(* CODESYS project SLL_IFM_CRXXXX_exported_from_plc.library
   Author: adam@sperrinlogic.com
   Version: 0.0.0.1
   Title: SLL_IFM_CRXXXX
   DefaultNamespace: SLL_IFM_CRXXXX
   Placeholder: SLL_IFM_CRXXXX
   Company: SLL

Project tree, tasks and I/O mapping:
  libraries: Util, 3.5.19.0 (System); Standard, 3.5.18.0 (System); ifmTypes, 1.9.6.0 (ifm electronic); ifmRawCAN, 4.0.3.0 (ifm electronic); ifmDeviceCR07nn, 1.2.2.0 (ifm electronic); SysTime, 3.5.17.0 (System); ifmIOcommon, 2.4.0.0 (ifm electronic); CmpSchedule, 3.5.17.0 (System); SysTypes Interfaces, * (System); SysTypes2 Interfaces, * (System); CmpIecTask, 3.5.19.0 (System); CmpErrors2 Interfaces, * (System); CmpErrors, 3.3.1.40 (System); SysFileAsync, 3.5.19.0 (System); SysTypes, 3.1.2.0 (System); SLL Common, 0.0.0.1 (SLL)
  Library Information/
    function IsLibReleased [ST]
    function GetLibVersionNumber [ST]
    function GetLibVersion [ST]
  data type PLC_CRXXXX_CAN_Status
  program PLC_CRXXXX_System_Udp [FBD]
  data type IFM_CRXXXX_System_STRUCT
  function block UDP_RX_CHECK_HB_FB [FBD]
  data type UDP_RX_STATS_HB_STRUCT
  data type IFM_HMI_Version_System_Header
  function block Get_Task_Info [ST]
  data type PLC_TASK_INFO_STRUCT
  program PLC_CRXXXX_System [FBD]
*)

// PLC_CRXXXX_CAN_Status
TYPE PLC_CRXXXX_CAN_Status :
STRUCT
	xError: BOOL;
	eDiagInfo: ifmTypes.DIAG_INFO;
	eBaudrate: ifmDevice.CAN_BAUDRATE;
	eBusState: ifmRCAN.BUS_STATE;
	uiErrorCntRx: UINT;
	uiErrorCntTx: UINT;
	xWarningRx: BOOL;
	xWarningTx: BOOL;
	udiCountRx: UDINT;
	usiBusLoad: USINT;
END_STRUCT
END_TYPE

// IFM_CRXXXX_System_STRUCT
TYPE IFM_CRXXXX_System_STRUCT :
STRUCT
	CycleCounter:DWORD;
	CycleFreq:REAL;
	CycleSecCounter:DWORD;
	CycleSecFreq:REAL;
	UpTimeMs:DWORD;
	VBB15_mV:UINT;
	VBB30_mV:UINT;
	PCB_Temp:INT;
	CPU_Temp:INT;
	TaskInfo: PLC_TASK_INFO_STRUCT;
	CAN0: PLC_CRXXXX_CAN_Status;
	CAN1: PLC_CRXXXX_CAN_Status;
	CAN2: PLC_CRXXXX_CAN_Status;
	CAN3: PLC_CRXXXX_CAN_Status;	
END_STRUCT
END_TYPE

// UDP_RX_STATS_HB_STRUCT
TYPE UDP_RX_STATS_HB_STRUCT :
STRUCT
	PLC_UpTimeMs:DINT;
	PLC_UpTimeMs_Last: DINT;
	PLC_UpTimeMs_Diff: DINT;
	
	Max_Diff_Value: DINT;	

	Error_LT_Count: DINT;
	Error_Diff_Count: DINT;
	Error_Frozen_Count: DINT;

	Warn_LT_Count: DINT;
	
	Warn_Diff_Count: DINT;
	Warn_Diff_TimeStamp: DWORD;
	Warn_Diff_Since: DWORD;

	Warn_Frozen_Count: DINT;

	Warn_Frozen_TimeStamp: DWORD;
	Warn_Frozen_Since: DWORD;	
END_STRUCT
END_TYPE

// IFM_HMI_Version_System_Header
TYPE IFM_HMI_Version_System_Header :
STRUCT
	TickMs: DWORD;
	Version_String: STRING(20);
	Version_Nums: ARRAY [0..3] OF WORD; 
	IO_Flags: WORD; // future use? special modes?
END_STRUCT
END_TYPE

// PLC_TASK_INFO_STRUCT
TYPE PLC_TASK_INFO_STRUCT :
STRUCT
    dwCycleTimeMainTask: DWORD;       
    dwCycleTimeSecTask: DWORD;       
    dwIntervalMainTask: DWORD;
    dwIntervalSecTask: DWORD;
    fMainTaskCpuLoad: REAL;
    fSecTaskCpuLoad: REAL;
    sNameMainTask: STRING(20);	
    sNameSecTask: STRING(20);	
END_STRUCT
END_TYPE

// Library Information/IsLibReleased
// This function has been automatically generated from the project information.
FUNCTION IsLibReleased : BOOL
VAR_INPUT
	
END_VAR

IsLibReleased := FALSE;

END_FUNCTION

// Library Information/GetLibVersionNumber
// This function has been automatically generated from the project information.
FUNCTION GetLibVersionNumber : DWORD
VAR_INPUT
	
END_VAR

GetLibVersionNumber := 1;

END_FUNCTION

// Library Information/GetLibVersion
// This function has been automatically generated from the project information.
FUNCTION GetLibVersion : VERSION
VAR_INPUT
	
END_VAR

GetLibVersion.uiMajor := 0;
GetLibVersion.uiMinor := 0;
GetLibVersion.uiServicePack := 0;
GetLibVersion.uiPatch := 1;

END_FUNCTION

// PLC_CRXXXX_System_Udp
PROGRAM PLC_CRXXXX_System_Udp

VAR_INPUT
	System: REFERENCE TO IFM_CRXXXX_System_STRUCT;
END_VAR

VAR	
	Cycle_Freq_FB: Cycle_Freq_REAL;
END_VAR

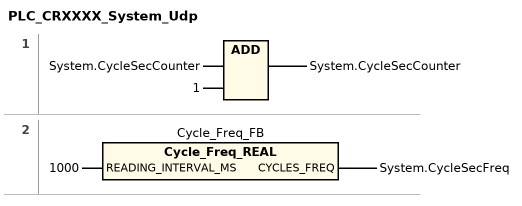
// NETWORK 1
System.CycleSecCounter := System.CycleSecCounter + 1;

// NETWORK 2
Cycle_Freq_FB(READING_INTERVAL_MS := 1000); // Cycle_Freq_REAL
System.CycleSecFreq := Cycle_Freq_FB.CYCLES_FREQ;

END_PROGRAM

// UDP_RX_CHECK_HB_FB
FUNCTION_BLOCK UDP_RX_CHECK_HB_FB
VAR_INPUT
	RESET: BOOL;	
	RESET_STATS: BOOL;
	RESET_ALARMS:BOOL;
	PlcTimeMs_Ip: DWORD;
	Moniotoring_Start_ms: DINT;	
	Warning_Diff_ms:DINT;
	Warning_Frozen_ms:DINT;
	Error_Diff_ms: DINT;
	Error_Frozen_ms: DINT;
	Error_Missing_ms: DINT;
	Error_Recovery_ms:DINT;
END_VAR
VAR_OUTPUT
	Monitoring: BOOL;	
	CommsError: BOOL;	
	Error_Missing: BOOL;
	Error_LessThan: BOOL;
	Error_Diff: BOOL;
	Error_Frozen: BOOL;
	Warning_Diff:BOOL;
	Warning_Frozen:BOOL;
	Unavail:BOOL:=TRUE;
END_VAR
VAR	
	TickMs: DWORD;
	TickMsWarmInit: DWORD;	
	
	RESET_Timestamp: DWORD;	
	RESET_Since_Ms: DWORD;
	
	Warning_Duration_Ms:DWORD:=1000;
	
	Warn_Frozen_TON:TON;
	
	Error_Missing_Active:BOOL;
	Error_Missing_Active_TON: TON;
	Error_Missing_SR: SR;
	Error_Missing_Reset_TON: TON;	
	Error_Missing_Set_TON: TON;
	
	Error_Frozen_Active: BOOL;
	Error_Frozen_Active_TON: TON;	
	Error_Frozen_SR: SR;
	Error_Frozen_Reset_TON: TON;
	Error_Frozen_Set_TON: TON;
	
	Error_Diff_Active: BOOL;
	Error_Diff_SR: SR;
	Error_Diff_Reset_TON: TON;
	Error_Diff_Set_TON: TON;
	
	Error_LessThan_Active: BOOL;
	Error_LessThan_SR: SR;
	Error_LessThan_Reset_TON: TON;	
	Error_LessThan_Set_TON: TON;
	Reset_Idle_TOF: TOF;
END_VAR

VAR_IN_OUT
	STATS: UDP_RX_STATS_HB_STRUCT;	
END_VAR
VAR // added by the converter: edge detectors and wires of the graphical bodies
    _w1, _w2 : BOOL;
    _rt1, _rt2, _rt3 : R_TRIG;
END_VAR

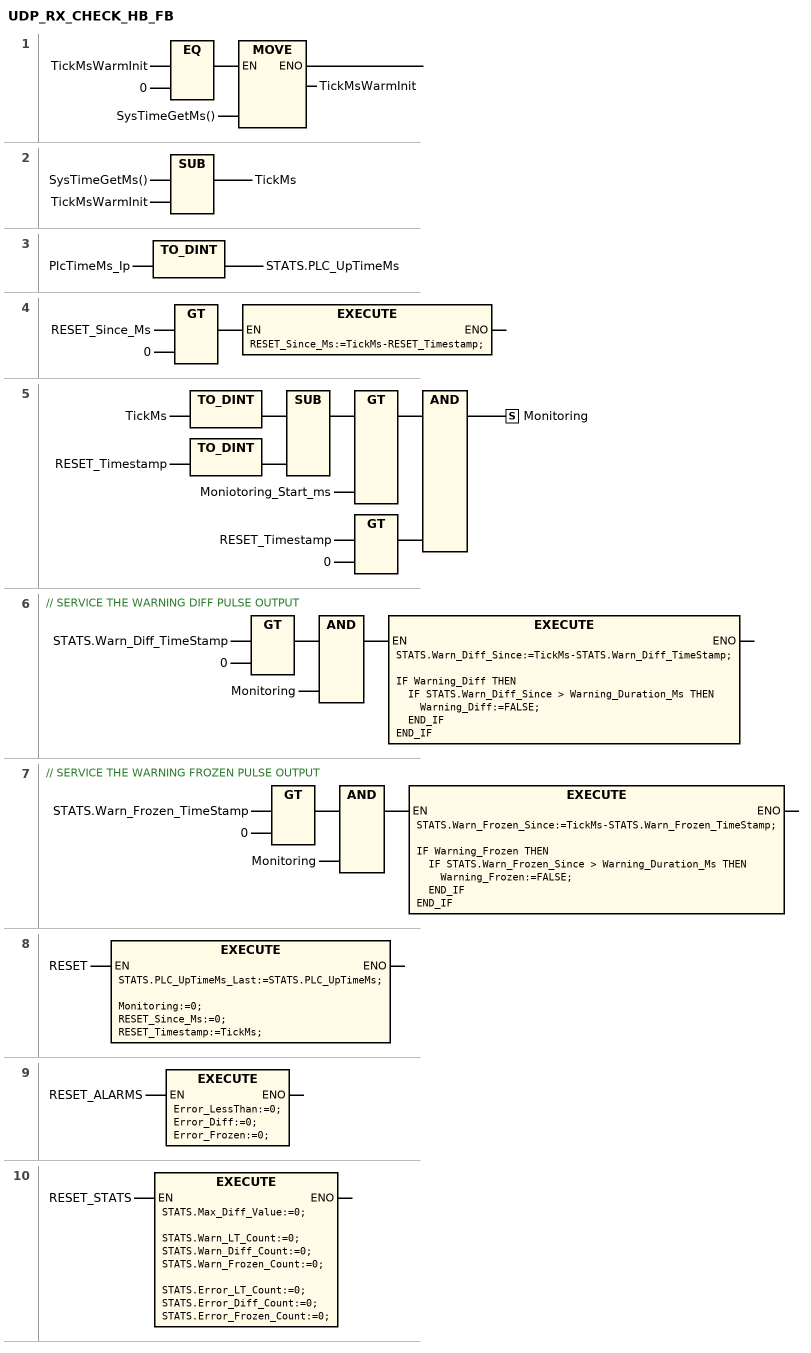
// NETWORK 1
IF TickMsWarmInit = 0 THEN TickMsWarmInit := SysTimeGetMs(); END_IF

// NETWORK 2
TickMs := (SysTimeGetMs()) - TickMsWarmInit;

// NETWORK 3
STATS.PLC_UpTimeMs := TO_DINT(PlcTimeMs_Ip);

// NETWORK 4
IF RESET_Since_Ms > 0 THEN RESET_Since_Ms:=TickMs-RESET_Timestamp; END_IF

// NETWORK 5
Monitoring S= TO_DINT(TickMs) - TO_DINT(RESET_Timestamp) > Moniotoring_Start_ms AND RESET_Timestamp > 0;

// NETWORK 6
// // SERVICE THE WARNING DIFF PULSE OUTPUT
IF STATS.Warn_Diff_TimeStamp > 0 AND Monitoring THEN
    STATS.Warn_Diff_Since:=TickMs-STATS.Warn_Diff_TimeStamp;
    
    IF Warning_Diff THEN
    	IF STATS.Warn_Diff_Since > Warning_Duration_Ms THEN
    		Warning_Diff:=FALSE;
    	END_IF
    END_IF
END_IF

// NETWORK 7
// // SERVICE THE WARNING FROZEN PULSE OUTPUT
IF STATS.Warn_Frozen_TimeStamp > 0 AND Monitoring THEN
    STATS.Warn_Frozen_Since:=TickMs-STATS.Warn_Frozen_TimeStamp;
    
    IF Warning_Frozen THEN
    	IF STATS.Warn_Frozen_Since > Warning_Duration_Ms THEN
    		Warning_Frozen:=FALSE;
    	END_IF
    END_IF
END_IF

// NETWORK 8
IF RESET THEN
    STATS.PLC_UpTimeMs_Last:=STATS.PLC_UpTimeMs;
    
    Monitoring:=0;
    RESET_Since_Ms:=0;
    RESET_Timestamp:=TickMs;
END_IF

// NETWORK 9
IF RESET_ALARMS THEN
    Error_LessThan:=0;
    Error_Diff:=0;
    Error_Frozen:=0;
END_IF

// NETWORK 10
IF RESET_STATS THEN
    STATS.Max_Diff_Value:=0;
    
    STATS.Warn_LT_Count:=0;
    STATS.Warn_Diff_Count:=0;
    STATS.Warn_Frozen_Count:=0;
    
    STATS.Error_LT_Count:=0;
    STATS.Error_Diff_Count:=0;
    STATS.Error_Frozen_Count:=0;
END_IF

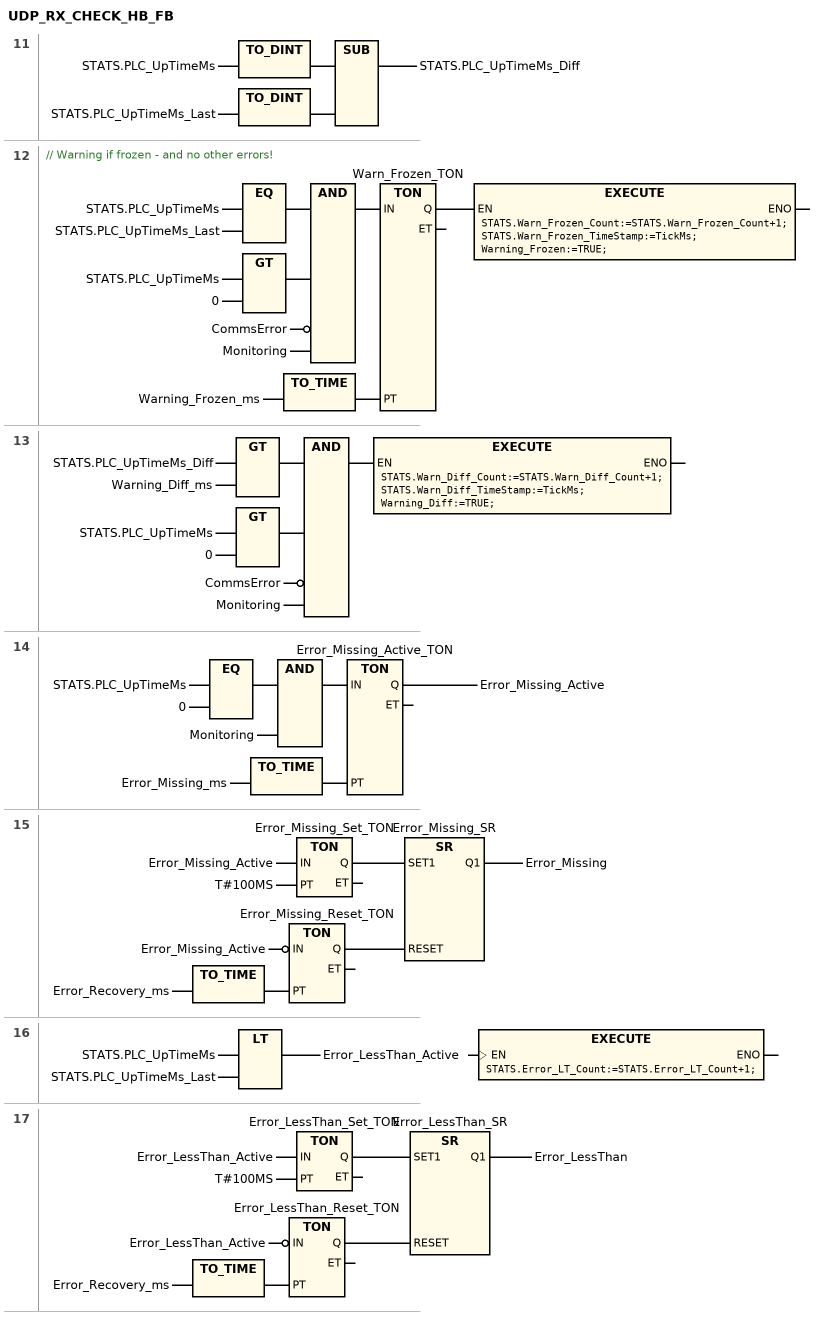
// NETWORK 11
STATS.PLC_UpTimeMs_Diff := TO_DINT(STATS.PLC_UpTimeMs) - TO_DINT(STATS.PLC_UpTimeMs_Last);

// NETWORK 12
// // Warning if frozen - and no other errors!
Warn_Frozen_TON(IN := STATS.PLC_UpTimeMs = STATS.PLC_UpTimeMs_Last AND STATS.PLC_UpTimeMs > 0 AND NOT CommsError AND Monitoring, PT := TO_TIME(Warning_Frozen_ms)); // TON
IF Warn_Frozen_TON.Q THEN
    STATS.Warn_Frozen_Count:=STATS.Warn_Frozen_Count+1;
    STATS.Warn_Frozen_TimeStamp:=TickMs;
    Warning_Frozen:=TRUE;
END_IF

// NETWORK 13
IF STATS.PLC_UpTimeMs_Diff > Warning_Diff_ms AND STATS.PLC_UpTimeMs > 0 AND NOT CommsError AND Monitoring THEN
    STATS.Warn_Diff_Count:=STATS.Warn_Diff_Count+1;
    STATS.Warn_Diff_TimeStamp:=TickMs;
    Warning_Diff:=TRUE;
END_IF

// NETWORK 14
Error_Missing_Active_TON(IN := STATS.PLC_UpTimeMs = 0 AND Monitoring, PT := TO_TIME(Error_Missing_ms)); // TON
Error_Missing_Active := Error_Missing_Active_TON.Q;

// NETWORK 15
Error_Missing_Set_TON(IN := Error_Missing_Active, PT := T#100MS); // TON
Error_Missing_Reset_TON(IN := NOT Error_Missing_Active, PT := TO_TIME(Error_Recovery_ms)); // TON
Error_Missing_SR(SET1 := Error_Missing_Set_TON.Q, RESET := Error_Missing_Reset_TON.Q); // SR
Error_Missing := Error_Missing_SR.Q1;

// NETWORK 16
_w1 := STATS.PLC_UpTimeMs < STATS.PLC_UpTimeMs_Last;
Error_LessThan_Active := _w1;
_rt1(CLK := _w1);
IF _rt1.Q THEN STATS.Error_LT_Count:=STATS.Error_LT_Count+1; END_IF

// NETWORK 17
Error_LessThan_Set_TON(IN := Error_LessThan_Active, PT := T#100MS); // TON
Error_LessThan_Reset_TON(IN := NOT Error_LessThan_Active, PT := TO_TIME(Error_Recovery_ms)); // TON
Error_LessThan_SR(SET1 := Error_LessThan_Set_TON.Q, RESET := Error_LessThan_Reset_TON.Q); // SR
Error_LessThan := Error_LessThan_SR.Q1;

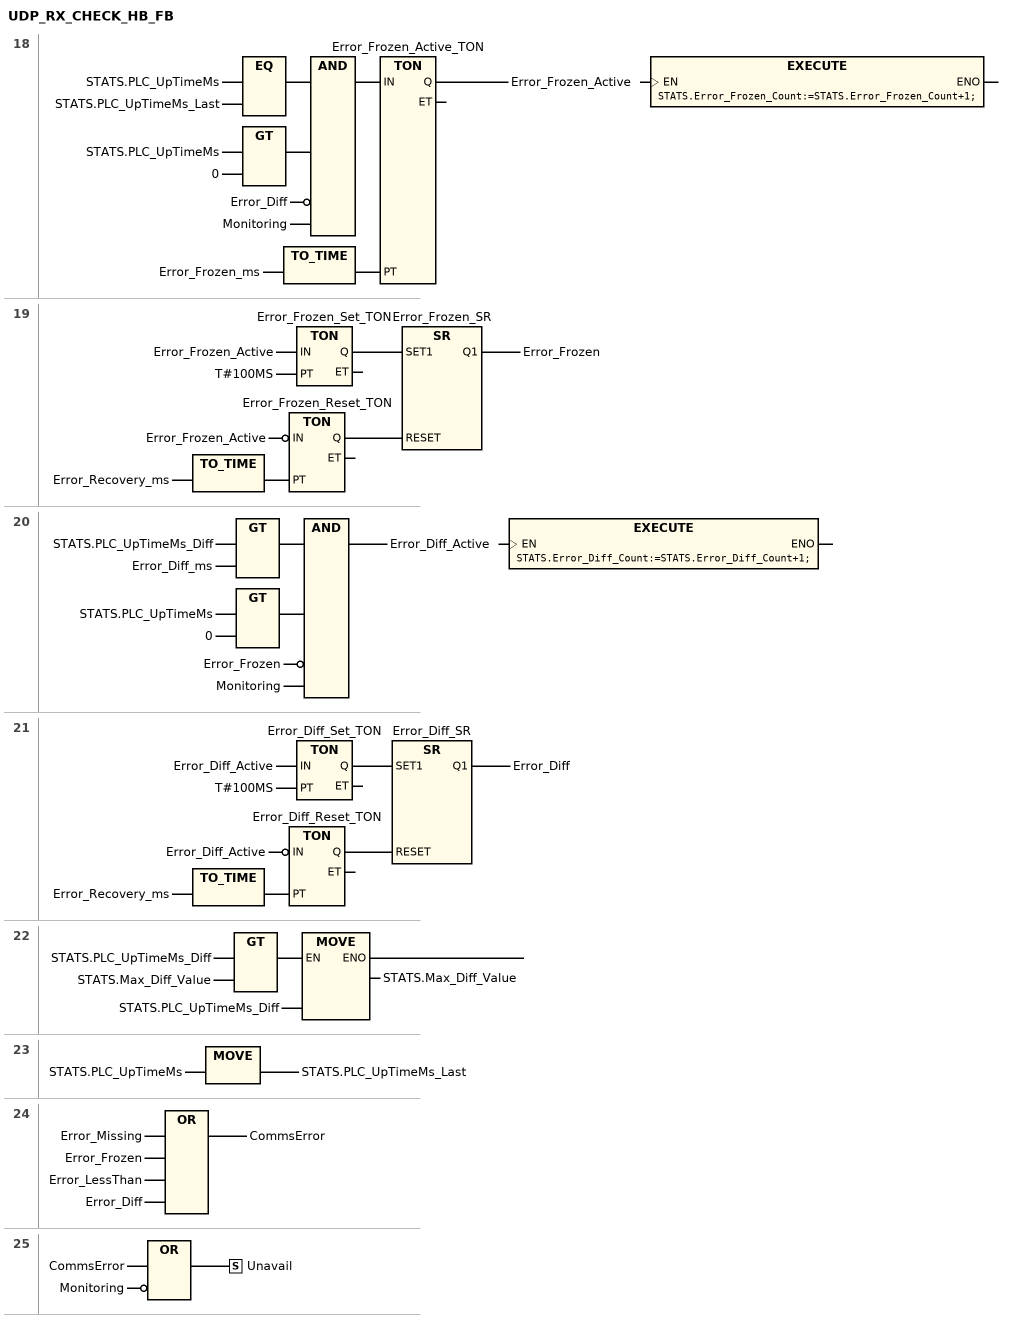
// NETWORK 18
Error_Frozen_Active_TON(IN := STATS.PLC_UpTimeMs = STATS.PLC_UpTimeMs_Last AND STATS.PLC_UpTimeMs > 0 AND NOT Error_Diff AND Monitoring, PT := TO_TIME(Error_Frozen_ms)); // TON
Error_Frozen_Active := Error_Frozen_Active_TON.Q;
_rt2(CLK := Error_Frozen_Active_TON.Q);
IF _rt2.Q THEN STATS.Error_Frozen_Count:=STATS.Error_Frozen_Count+1; END_IF

// NETWORK 19
Error_Frozen_Set_TON(IN := Error_Frozen_Active, PT := T#100MS); // TON
Error_Frozen_Reset_TON(IN := NOT Error_Frozen_Active, PT := TO_TIME(Error_Recovery_ms)); // TON
Error_Frozen_SR(SET1 := Error_Frozen_Set_TON.Q, RESET := Error_Frozen_Reset_TON.Q); // SR
Error_Frozen := Error_Frozen_SR.Q1;

// NETWORK 20
_w2 := STATS.PLC_UpTimeMs_Diff > Error_Diff_ms AND STATS.PLC_UpTimeMs > 0 AND NOT Error_Frozen AND Monitoring;
Error_Diff_Active := _w2;
_rt3(CLK := _w2);
IF _rt3.Q THEN STATS.Error_Diff_Count:=STATS.Error_Diff_Count+1; END_IF

// NETWORK 21
Error_Diff_Set_TON(IN := Error_Diff_Active, PT := T#100MS); // TON
Error_Diff_Reset_TON(IN := NOT Error_Diff_Active, PT := TO_TIME(Error_Recovery_ms)); // TON
Error_Diff_SR(SET1 := Error_Diff_Set_TON.Q, RESET := Error_Diff_Reset_TON.Q); // SR
Error_Diff := Error_Diff_SR.Q1;

// NETWORK 22
IF STATS.PLC_UpTimeMs_Diff > STATS.Max_Diff_Value THEN STATS.Max_Diff_Value := STATS.PLC_UpTimeMs_Diff; END_IF

// NETWORK 23
STATS.PLC_UpTimeMs_Last := STATS.PLC_UpTimeMs;

// NETWORK 24
CommsError := Error_Missing OR Error_Frozen OR Error_LessThan OR Error_Diff;

// NETWORK 25
Unavail S= CommsError OR NOT Monitoring;

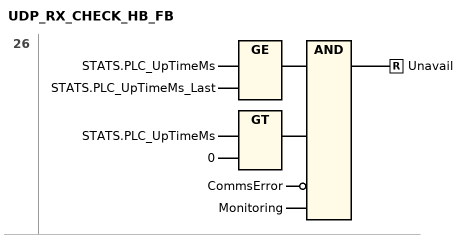
// NETWORK 26
Unavail R= STATS.PLC_UpTimeMs >= STATS.PLC_UpTimeMs_Last AND STATS.PLC_UpTimeMs > 0 AND NOT CommsError AND Monitoring;

END_FUNCTION_BLOCK

// Get_Task_Info
FUNCTION_BLOCK Get_Task_Info
VAR_INPUT
	sample_rate_tm:DWORD:=500;
END_VAR
VAR
    hFirstTask, hSecTask                       :    SysTypes.RTS_IEC_HANDLE;
    iecResult                                  :    SysTypes.RTS_IEC_RESULT;
    sAppName                                   :    STRING := 'Application';
    pIecInfo                                   :    POINTER TO CmpIecTask.Task_Info2;
	
	last_sample_ms: DWORD;
	diff_ms: DWORD;	
END_VAR

VAR_OUTPUT
	TaskInfo: PLC_TASK_INFO_STRUCT;
END_VAR

diff_ms := SysTimeGetMs() - last_sample_ms;

IF diff_ms < sample_rate_tm THEN
	RETURN;
END_IF

hFirstTask := CmpIecTask.IecTaskGetFirst(pszAppName := ADR(sAppName), pResult := ADR(iecResult));

IF ((hFirstTask <> SysTypes.RTS_INVALID_HANDLE) AND (iecResult = CmpErrors.Errors.ERR_OK)) THEN
    pIecInfo := CmpIecTask.IecTaskGetInfo3(hIecTask := hFirstTask, pResult := ADR(iecResult));
    TaskInfo.dwIntervalMainTask := pIecInfo^.dwInterval;
    TaskInfo.dwCycleTimeMainTask := pIecInfo^.dwCycleTime;
    TaskInfo.sNameMainTask := pIecInfo^.pszName^;
	
    hSecTask := IecTaskGetNext(pszAppName := ADR(sAppName), hPrevIecTask := hFirstTask, pResult := ADR(iecResult));
    IF ((hSecTask <> SysTypes.RTS_INVALID_HANDLE) AND (iecResult = CmpErrors.Errors.ERR_OK)) THEN
        pIecInfo := CmpIecTask.IecTaskGetInfo3(hIecTask := hSecTask, pResult := ADR(iecResult));
        TaskInfo.dwIntervalSecTask := pIecInfo^.dwInterval;
        TaskInfo.dwCycleTimeSecTask := pIecInfo^.dwCycleTime;
        TaskInfo.sNameSecTask := pIecInfo^.pszName^;
    END_IF
END_IF

TaskInfo.fMainTaskCpuLoad:=TO_REAL(TaskInfo.dwCycleTimeMainTask*100)/TO_REAL(TaskInfo.dwIntervalMainTask);
TaskInfo.fSecTaskCpuLoad:=TO_REAL(TaskInfo.dwCycleTimeSecTask*100)/TO_REAL(TaskInfo.dwIntervalSecTask);

END_FUNCTION_BLOCK

// PLC_CRXXXX_System
PROGRAM PLC_CRXXXX_System

VAR_INPUT
	System: REFERENCE TO IFM_CRXXXX_System_STRUCT;
END_VAR

VAR	
	Temperature_PCB_FB: ifmIOcommon.Temperature;
	Temperature_CPU_FB: ifmIOcommon.Temperature;	
	SystemSupply_VBB30_FB: ifmIOcommon.SystemSupply;
	SystemSupply_VBB15_FB: ifmIOcommon.SystemSupply;
	Cycle_Freq_FB: Cycle_Freq_REAL;
	CAN0_Status:  ifmRCAN.CAN_Status;
	CAN1_Status: ifmRCAN.CAN_Status;
	CAN2_Status: ifmRCAN.CAN_Status;
	CAN3_Status: ifmRCAN.CAN_Status;
	
	TickMsWarmInit:DWORD;
	Get_Task_Info_FB: Get_Task_Info;
END_VAR
VAR // added by the converter: edge detectors and wires of the graphical bodies
    _rt1 : R_TRIG;
END_VAR

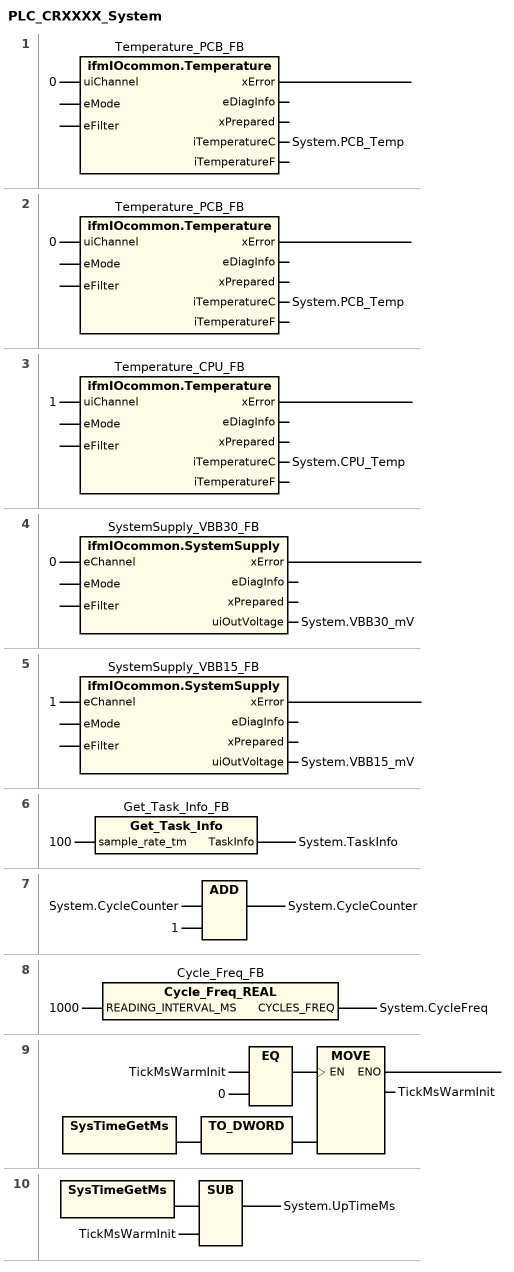
// NETWORK 1
Temperature_PCB_FB(uiChannel := 0, iTemperatureC => System.PCB_Temp); // ifmIOcommon.Temperature

// NETWORK 2
Temperature_PCB_FB(uiChannel := 0, iTemperatureC => System.PCB_Temp); // ifmIOcommon.Temperature

// NETWORK 3
Temperature_CPU_FB(uiChannel := 1, iTemperatureC => System.CPU_Temp); // ifmIOcommon.Temperature

// NETWORK 4
SystemSupply_VBB30_FB(eChannel := 0, uiOutVoltage => System.VBB30_mV); // ifmIOcommon.SystemSupply

// NETWORK 5
SystemSupply_VBB15_FB(eChannel := 1, uiOutVoltage => System.VBB15_mV); // ifmIOcommon.SystemSupply

// NETWORK 6
Get_Task_Info_FB(sample_rate_tm := 100); // Get_Task_Info
System.TaskInfo := Get_Task_Info_FB.TaskInfo;

// NETWORK 7
System.CycleCounter := System.CycleCounter + 1;

// NETWORK 8
Cycle_Freq_FB(READING_INTERVAL_MS := 1000); // Cycle_Freq_REAL
System.CycleFreq := Cycle_Freq_FB.CYCLES_FREQ;

// NETWORK 9
_rt1(CLK := TickMsWarmInit = 0);
IF _rt1.Q THEN TickMsWarmInit := TO_DWORD(SysTimeGetMs()); END_IF

// NETWORK 10
System.UpTimeMs := SysTimeGetMs() - TickMsWarmInit;

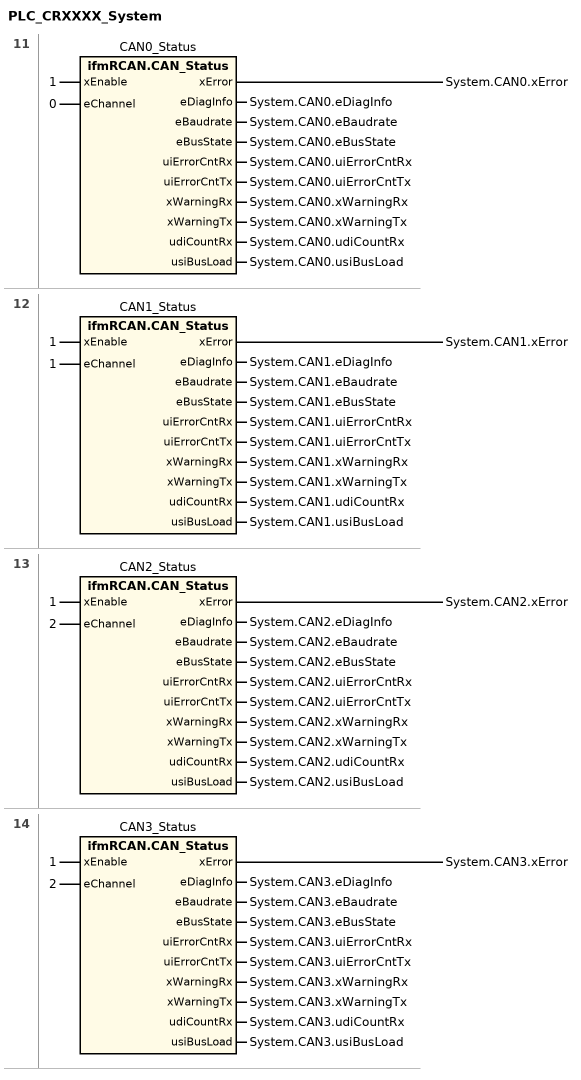
// NETWORK 11
CAN0_Status(
    xEnable := 1,
    eChannel := 0,
    eDiagInfo => System.CAN0.eDiagInfo,
    eBaudrate => System.CAN0.eBaudrate,
    eBusState => System.CAN0.eBusState,
    uiErrorCntRx => System.CAN0.uiErrorCntRx,
    uiErrorCntTx => System.CAN0.uiErrorCntTx,
    xWarningRx => System.CAN0.xWarningRx,
    xWarningTx => System.CAN0.xWarningTx,
    udiCountRx => System.CAN0.udiCountRx,
    usiBusLoad => System.CAN0.usiBusLoad); // ifmRCAN.CAN_Status
System.CAN0.xError := CAN0_Status.xError;

// NETWORK 12
CAN1_Status(
    xEnable := 1,
    eChannel := 1,
    eDiagInfo => System.CAN1.eDiagInfo,
    eBaudrate => System.CAN1.eBaudrate,
    eBusState => System.CAN1.eBusState,
    uiErrorCntRx => System.CAN1.uiErrorCntRx,
    uiErrorCntTx => System.CAN1.uiErrorCntTx,
    xWarningRx => System.CAN1.xWarningRx,
    xWarningTx => System.CAN1.xWarningTx,
    udiCountRx => System.CAN1.udiCountRx,
    usiBusLoad => System.CAN1.usiBusLoad); // ifmRCAN.CAN_Status
System.CAN1.xError := CAN1_Status.xError;

// NETWORK 13
CAN2_Status(
    xEnable := 1,
    eChannel := 2,
    eDiagInfo => System.CAN2.eDiagInfo,
    eBaudrate => System.CAN2.eBaudrate,
    eBusState => System.CAN2.eBusState,
    uiErrorCntRx => System.CAN2.uiErrorCntRx,
    uiErrorCntTx => System.CAN2.uiErrorCntTx,
    xWarningRx => System.CAN2.xWarningRx,
    xWarningTx => System.CAN2.xWarningTx,
    udiCountRx => System.CAN2.udiCountRx,
    usiBusLoad => System.CAN2.usiBusLoad); // ifmRCAN.CAN_Status
System.CAN2.xError := CAN2_Status.xError;

// NETWORK 14
CAN3_Status(
    xEnable := 1,
    eChannel := 2,
    eDiagInfo => System.CAN3.eDiagInfo,
    eBaudrate => System.CAN3.eBaudrate,
    eBusState => System.CAN3.eBusState,
    uiErrorCntRx => System.CAN3.uiErrorCntRx,
    uiErrorCntTx => System.CAN3.uiErrorCntTx,
    xWarningRx => System.CAN3.xWarningRx,
    xWarningTx => System.CAN3.xWarningTx,
    udiCountRx => System.CAN3.udiCountRx,
    usiBusLoad => System.CAN3.usiBusLoad); // ifmRCAN.CAN_Status
System.CAN3.xError := CAN3_Status.xError;

END_PROGRAM
